// TIA Portal V14 program export: 1 tag tables, 0 data types, 0 data blocks, 4 code blocks (in call order from the OBs), 0 instance data blocks

VAR_GLOBAL   // PLC tag table "IO_Tags"
   DI_Motor1_Feedback AT %I0.0 : Bool;   // Motor 1 running feedback
   DI_Motor2_Feedback AT %I0.1 : Bool;   // Motor 2 running feedback
   DI_Emergency_Stop AT %I0.2 : Bool;   // Emergency stop button
   AI_Temperature AT %IW64 : Int;   // Temperature sensor analog input
   DO_Motor1_Run AT %Q0.0 : Bool;   // Motor 1 run command
   DO_Motor2_Run AT %Q0.1 : Bool;   // Motor 2 run command
   DO_Valve1 AT %Q0.2 : Bool;   // Valve 1 control
   AO_Speed_Ref AT %QW64 : Int;   // Speed reference analog output
END_VAR

ORGANIZATION_BLOCK "Main"   // OB1, SCL
// stored: AutoNumber true
BEGIN
END_ORGANIZATION_BLOCK

ORGANIZATION_BLOCK "Startup"   // OB100, SCL
// stored: AutoNumber true
BEGIN
END_ORGANIZATION_BLOCK

FUNCTION_BLOCK "FB_MotorControl"   // FB1, SCL
// stored: AutoNumber true
BEGIN
END_FUNCTION_BLOCK

FUNCTION "FC_DataProcess" : Void   // FC1, SCL
// stored: AutoNumber true
BEGIN
END_FUNCTION
